FUNCTION_BLOCK FB_MachinePreparation
VAR_INPUT
    // 自动启动协调器或WPF一键整机准备请求。
    // 只受理FALSE→TRUE上升沿。
    bStart : BOOL;

    // Stop、整机故障或流程中止。
    bAbort : BOOL;

    // 故障复位脉冲。
    bReset : BOOL;

    stConfig : ST_MachinePreparationConfig;
END_VAR

VAR_IN_OUT
    aAxes : ARRAY[1..GVL_Constants.cMaxAxisCount]
            OF ST_AxisInterface;
	// 复用MAIN中COM3唯一的自动动作实例。
    // 禁止在准备流程中重新创建FB_GripperAction实例。
    ioGripperAction : FB_GripperAction;
	// 复用MAIN中COM4唯一的自动动作实例。
    ioAdjustGripperAction : FB_GripperAction;

    // COM3夹爪统一接口。
    ioGripper : ST_GripperInterface;
	// COM4调整夹爪统一接口。
    ioAdjustGripper : ST_GripperInterface;
END_VAR

VAR_OUTPUT
    bBusy       : BOOL;
    bDone       : BOOL;
    bError      : BOOL;
    bErrorPulse : BOOL;
    bTimeout    : BOOL;

    uiErrorAxis : UINT;
    udiErrorCode : UDINT;

    eStep : E_MachinePreparationStep :=
        E_MachinePreparationStep.Idle;
END_VAR

VAR
    trigStart : R_TRIG;

    fbReadyTimeout  : TON;
    fbMotionTimeout : TON;
    // 准备私有Tray恢复上下文，每次Start/Stop/Fault均清理。
    eTrayRecoveryStep : E_MachinePreparationStep := E_MachinePreparationStep.TrayWaitForkStable;
    nRecoveryTargetLayer : DINT;
    nRecoveryIndex : DINT;
    nRecoveryMatchCount : DINT;
    bTrayRecoverySelected : BOOL;
    bTrayRecoveryActive : BOOL;
    bRecoveryClassC : BOOL;
    bRecoveryRackPermit : BOOL;
    fbTrayRecoveryTimeout : TON;
    fbTrayReleaseTimeout : TON;
    fbTrayReleaseStable : TON;
    bReleaseConditions : BOOL;
    fbForkStable : TON;
    bForkCandidateInitialized : BOOL;
    bForkCandidate : BOOL;
    bForkStable : BOOL;
    bForkStableValid : BOOL;
    aRecoveryLevelTimer : ARRAY[1..5] OF TON;
    aRecoveryLevelInitialized : ARRAY[1..5] OF BOOL;
    aRecoveryLevelCandidate : ARRAY[1..5] OF BOOL;
    aRecoveryLevelStable : ARRAY[1..5] OF BOOL;
    aRecoveryLevelStableValid : ARRAY[1..5] OF BOOL;
    bRecoveryAllLevelsStable : BOOL;
    bNonTrayStandbyDone : BOOL;

    uiItem : DINT;
    uiAxis : UINT;
    bAllAxesReady : BOOL;

    // 各轴命令已发出锁存
    bTrayXIssued       : BOOL;
    bTrayZIssued       : BOOL;
    bDamperXIssued     : BOOL;
    bDamperYIssued     : BOOL;
    bDamperZIssued     : BOOL;
    bRotationIssued    : BOOL;
    bClampIssued       : BOOL;
    bTurntableIssued   : BOOL;
	bAdjustmentXIssued : BOOL;
	bAdjustmentYIssued : BOOL;
	bAdjustmentZIssued : BOOL;
    bScrewYIssued      : BOOL;
    bScrewZIssued      : BOOL;

    // 各轴到位锁存
    bTrayXDone       : BOOL;
    bTrayZDone       : BOOL;
    bDamperXDone     : BOOL;
    bDamperYDone     : BOOL;
    bDamperZDone     : BOOL;
    bRotationDone    : BOOL;
    bClampDone       : BOOL;
    bTurntableDone   : BOOL;
	bAdjustmentXDone : BOOL;
	bAdjustmentYDone : BOOL;
	bAdjustmentZDone : BOOL;
    bScrewYDone      : BOOL;
    bScrewZDone      : BOOL;
	
	// 机构准备阶段的COM3张开请求。
    // 在MoveToStandby期间保持TRUE，完成后恢复FALSE。
    bGripperOpenExecute : BOOL;

    // COM3夹爪已经张开完成的锁存状态。
    bGripperOpenDone : BOOL;
    bGripperEnableExecute : BOOL;
    bGripperEnableDone : BOOL; // 本次准备Enable写事务完成，不是硬件使能状态
    bGripperEnableReleasePending : BOOL;
    eGripperPreparationCommand : E_GripperCommand;

	// AdjustmentZ处于安全位置后执行COM4闭合。
	bAdjustGripperCloseExecute : BOOL;
	bAdjustGripperCloseDone : BOOL;
    bAdjustGripperEnableExecute : BOOL;
    bAdjustGripperEnableDone : BOOL;
    bAdjustGripperEnableReleasePending : BOOL;
    eAdjustGripperPreparationCommand : E_GripperCommand;
	bAdjustGripperReady : BOOL;
	liAdjustGripperPositionError : LINT;
END_VAR

//==============================================================
// 1. 请求及定时器
//==============================================================
trigStart(CLK := bStart);

fbReadyTimeout(
    IN := (eStep = E_MachinePreparationStep.WaitAxesReady)
          AND NOT bAbort,
    PT := stConfig.tReadyTimeout
);

bErrorPulse := FALSE;
// 默认不请求夹爪动作。
// 只有MoveToStandby步骤尚未完成张开时才置TRUE。
bGripperOpenExecute := FALSE;
bAdjustGripperCloseExecute := FALSE;

bGripperEnableExecute := FALSE;
bAdjustGripperEnableExecute := FALSE;
eGripperPreparationCommand := E_GripperCommand.Open;
eAdjustGripperPreparationCommand := E_GripperCommand.Close;

// COM4准备完成必须由真实状态共同确认，不能只依赖动作完成握手。
liAdjustGripperPositionError :=
    DINT_TO_LINT(ioAdjustGripper.Feedback.diActualPosition)
    - DINT_TO_LINT(ioAdjustGripper.Set.diClosePosition);
IF liAdjustGripperPositionError < 0 THEN
    liAdjustGripperPositionError := -liAdjustGripperPositionError;
END_IF;

bAdjustGripperReady :=
    ioAdjustGripper.State.bSimulationActive
    OR (ioAdjustGripper.Feedback.bOnline
    AND NOT ioAdjustGripper.Feedback.bCommFault
    AND ioAdjustGripper.Feedback.bFaultCodeValid
    AND NOT ioAdjustGripper.Feedback.bFault
    AND NOT ioAdjustGripper.State.bBusy
    AND NOT ioAdjustGripper.Feedback.bBusy
    AND ioAdjustGripper.Feedback.bPositionValid
    AND ioAdjustGripper.Feedback.bCurrentValid
    AND
    (
        liAdjustGripperPositionError
        <= DINT_TO_LINT(ioAdjustGripper.Set.diPositionTolerance)
    )
    AND ioAdjustGripper.Feedback.bClosed);

// 原超时仍保护全部非Tray准备机构；有盘回库由独立总超时保护。
bNonTrayStandbyDone := bDamperXDone AND bDamperYDone AND bDamperZDone
              AND bRotationDone AND bClampDone AND bTurntableDone
              AND bAdjustmentXDone AND bAdjustmentYDone AND bAdjustmentZDone
              AND bScrewYDone AND bScrewZDone
              AND bGripperOpenDone AND bAdjustGripperCloseDone AND bAdjustGripperReady;
fbMotionTimeout(
    IN := (eStep = E_MachinePreparationStep.MoveToStandby)
        AND NOT bAbort
        AND (NOT bNonTrayStandbyDone
            OR (NOT bTrayRecoverySelected AND NOT (bTrayXDone AND bTrayZDone))),
    PT := stConfig.tMotionTimeout
);

//==============================================================
// 2. Preparation命令脉冲默认清除
// 只处理当前十根已明确准备位置的自动流程轴。
//==============================================================
FOR uiItem := LOWER_BOUND(GVL_AxisIndex.AutoProcessAxes, 1) TO UPPER_BOUND(GVL_AxisIndex.AutoProcessAxes, 1) DO
    uiAxis := GVL_AxisIndex.AutoProcessAxes[uiItem];

    aAxes[uiAxis].PreparationCmd.bMoveAbs := FALSE;
    aAxes[uiAxis].PreparationCmd.bMoveRel := FALSE;
    aAxes[uiAxis].PreparationCmd.bJogPos := FALSE;
    aAxes[uiAxis].PreparationCmd.bJogNeg := FALSE;
    aAxes[uiAxis].PreparationCmd.bStop := FALSE;
    aAxes[uiAxis].PreparationCmd.bTorqueControl := FALSE;
END_FOR;


//==============================================================
// 3. 故障复位和Abort
//
// 复位优先于Abort：准备故障会使整机进入Fault，
// 此时bAbort必然为TRUE，因此必须允许复位先清除本FB故障。
//==============================================================
IF bReset THEN
    bBusy := FALSE;
    bDone := FALSE;
    bError := FALSE;
    bTimeout := FALSE;

    uiErrorAxis := 0;
    udiErrorCode := TO_UDINT(E_MachinePreparationErrorCode.None);

    M_ResetProgress();

    eStep := E_MachinePreparationStep.Idle;

ELSIF bAbort THEN
    bBusy := FALSE;
    bDone := FALSE;

    M_ResetProgress();

    // 如果本FB本身已经报错，保持Error状态，
    // 便于故障诊断和后续统一复位。
    IF bError THEN
        eStep := E_MachinePreparationStep.Error;
    ELSE
        eStep := E_MachinePreparationStep.Idle;
    END_IF;

ELSE
    // 仅Done收到新请求时失效旧完成状态；Start撤销不清除本周期Done。
    // 同一扫描复用Idle中的配置检查和M_ResetProgress，不复制准备状态机。
    IF (eStep = E_MachinePreparationStep.Done) AND trigStart.Q THEN
        bDone := FALSE;
        eStep := E_MachinePreparationStep.Idle;
    END_IF;

    CASE eStep OF

        //======================================================
        // 等待启动
        //======================================================
        E_MachinePreparationStep.Idle:
            bBusy := FALSE;

            IF trigStart.Q THEN
                bDone := FALSE;
                bError := FALSE;
                bTimeout := FALSE;
                uiErrorAxis := 0;
                udiErrorCode := TO_UDINT(E_MachinePreparationErrorCode.None);

                M_ResetProgress();

                // 确认十根准备轴均已配置。
                FOR uiItem := 1 TO
                    UPPER_BOUND(GVL_AxisIndex.AutoProcessAxes, 1)
                DO
                    uiAxis :=
                        GVL_AxisIndex.AutoProcessAxes[uiItem];

                    IF NOT GVL_AxisConfig.AxisLimits[
                        uiAxis
                    ].bConfigured THEN
                        bError := TRUE;
                        bErrorPulse := TRUE;
                        uiErrorAxis := uiAxis;
                        udiErrorCode := TO_UDINT(E_MachinePreparationErrorCode.AxisNotConfigured);
                        eStep :=
                            E_MachinePreparationStep.Error;
                        EXIT;
                    END_IF;
                END_FOR;

                IF NOT bError THEN
                    bBusy := TRUE;
                    eStep :=
                        E_MachinePreparationStep.WaitAxesReady;
                END_IF;
            END_IF;


        //======================================================
        // 请求轴使能并等待全部Ready
        //======================================================
        E_MachinePreparationStep.WaitAxesReady:
            bBusy := TRUE;
            bAllAxesReady := TRUE;
            uiErrorAxis := 0;

            FOR uiItem := 1 TO
                UPPER_BOUND(GVL_AxisIndex.AutoProcessAxes, 1)
            DO
                uiAxis :=
                    GVL_AxisIndex.AutoProcessAxes[uiItem];

                IF aAxes[uiAxis].Alarm.bError THEN
                    bError := TRUE;
                    bErrorPulse := TRUE;
                    uiErrorAxis := uiAxis;

                    IF aAxes[uiAxis].Alarm.nErrorID <> 0 THEN
                        udiErrorCode :=
                            aAxes[uiAxis].Alarm.nErrorID;
                    ELSE
                        udiErrorCode := TO_UDINT(E_MachinePreparationErrorCode.AxisAlarmBase)
                            + UINT_TO_UDINT(uiAxis);
                    END_IF;

                    eStep :=
                        E_MachinePreparationStep.Error;
                    EXIT;
                END_IF;

                // Clamping必须先由真实6061确认已经恢复CSP。
                // 若PLC重新激活后驱动仍残留CST，则通过既有MC_Stop
                // 恢复边界请求退出；6061不是8时绝不发布准备运动。
                IF
                    (uiAxis = GVL_AxisIndex.Clamping)
                    AND
                    (
                        aAxes[uiAxis].State.eControlMode
                        <> E_AxisControlMode.Position
                    )
                THEN
                    aAxes[uiAxis].PreparationCmd.bTorqueControl := FALSE;
                    aAxes[uiAxis].PreparationCmd.bStop := TRUE;
                    bAllAxesReady := FALSE;

                    IF uiErrorAxis = 0 THEN
                        uiErrorAxis := uiAxis;
                    END_IF;
                END_IF;

                IF NOT aAxes[uiAxis].State.bReady THEN
                    bAllAxesReady := FALSE;

                    IF uiErrorAxis = 0 THEN
                        uiErrorAxis := uiAxis;
                    END_IF;
                END_IF;
            END_FOR;

            IF eStep <> E_MachinePreparationStep.Error THEN
                IF bAllAxesReady THEN
                    uiErrorAxis := 0;
                    eStep :=
                        E_MachinePreparationStep.MoveToStandby;

                ELSIF fbReadyTimeout.Q THEN
                    bError := TRUE;
                    bTimeout := TRUE;
                    bErrorPulse := TRUE;
                    udiErrorCode := TO_UDINT(E_MachinePreparationErrorCode.AxisReadyTimeout);
                    eStep :=
                        E_MachinePreparationStep.Error;
                END_IF;
            END_IF;


        //======================================================
        // 整机准备位置运动
        //
        // 三条机械分支并行执行：
        // A. TrayX安全后允许TrayZ
        // B. DamperZ安全后允许DamperXY和Rotation
        // C. ScrewdriverZ安全后允许夹紧松开和Y回零，
        //    夹紧松开后允许转台回零
        //======================================================
        E_MachinePreparationStep.MoveToStandby:
            bBusy := TRUE;
			
			//======================================================
			// COM3夹爪准备动作
			//
			// 与DamperZ抬升同时启动，不需要等待DamperZ到位。
			// bExecute保持TRUE，直到FB_GripperAction返回Done。
			//======================================================
            // 同一路复用唯一Action：Enable完成后FALSE释放，Idle后才发位置动作。
            IF NOT bGripperEnableDone THEN
                eGripperPreparationCommand := E_GripperCommand.Enable;
                bGripperEnableExecute := TRUE;
                IF ioGripperAction.bError THEN
                    bGripperEnableExecute := FALSE;
                    bError := TRUE;
                    bErrorPulse := TRUE;
                    uiErrorAxis := 0;
                    udiErrorCode := TO_UDINT(E_MachinePreparationErrorCode.DamperGripperEnableFailed);
                    // 具体底层原因仍保留在Action/AutoFeedback中。
                    eStep := E_MachinePreparationStep.Error;
                ELSIF ioGripperAction.bDone THEN
                    bGripperEnableDone := TRUE;
                    bGripperEnableReleasePending := TRUE;
                    bGripperEnableExecute := FALSE;
                END_IF;
            ELSIF bGripperEnableReleasePending THEN
                IF ioGripperAction.eStep = E_GripperActionStep.Idle THEN
                    bGripperEnableReleasePending := FALSE;
                END_IF;
            ELSIF NOT bGripperOpenDone THEN
                bGripperOpenExecute := TRUE;
			
				// FB_GripperAction在MAIN中的调用结果会跨扫描周期更新。
				IF ioGripperAction.bError THEN
					// COM3张开失败，机构准备失败。
					bGripperOpenExecute := FALSE;
			
					bError := TRUE;
					bErrorPulse := TRUE;
					uiErrorAxis := 0; // 夹爪不是NC轴，所以轴号为0。
			
					// 优先保留下层夹爪错误码，便于追踪具体动作失败原因。
					IF ioGripperAction.udErrorCode <> TO_UDINT(E_GripperErrorCode.None) THEN
						udiErrorCode := ioGripperAction.udErrorCode;
					ELSE
						udiErrorCode := TO_UDINT(E_MachinePreparationErrorCode.GripperOpenFailed);
					END_IF;
			
					eStep := E_MachinePreparationStep.Error;
			
				ELSIF ioGripperAction.bDone THEN
					// 张开完成后锁存，避免重复下发Open。
					bGripperOpenDone := TRUE;
					bGripperOpenExecute := FALSE;
				END_IF;
			END_IF;
            // Tray先等待Fork稳定，再执行原无盘路径或A/B/C恢复。
			M_PrepareTray(
				ioAxes := aAxes
			);
            // 其它机构继续保持原有并行准备时序。
            IF NOT bDamperZDone THEN
                bDamperZDone := M_MoveAxisAbsolute(
                    fTarget := stConfig.fDamperZStandby,
                    fVelocity := stConfig.fDamperVelocity,
                    fTolerance := stConfig.fLinearTolerance,
                    uiAxisIndex := GVL_AxisIndex.DamperZ,
                    ioIssued := bDamperZIssued,
                    ioAxis := aAxes[GVL_AxisIndex.DamperZ]
                );
            END_IF;

            IF NOT bScrewZDone THEN
                bScrewZDone := M_MoveAxisAbsolute(
                    fTarget := stConfig.fScrewdriverZSafe,
                    fVelocity := stConfig.fScrewdriverVelocity,
                    fTolerance := stConfig.fLinearTolerance,
                    uiAxisIndex := GVL_AxisIndex.ScrewdriverZ,
                    ioIssued := bScrewZIssued,
                    ioAxis := aAxes[GVL_AxisIndex.ScrewdriverZ]
                );
            END_IF;


            // DamperZ在110mm后，允许XY及旋转轴并行回位。
            IF bDamperZDone THEN
                IF NOT bDamperXDone THEN
                    bDamperXDone := M_MoveAxisAbsolute(
                        fTarget := stConfig.fDamperXStandby,
                        fVelocity := stConfig.fDamperVelocity,
                        fTolerance := stConfig.fLinearTolerance,
                        uiAxisIndex := GVL_AxisIndex.DamperX,
                        ioIssued := bDamperXIssued,
                        ioAxis := aAxes[GVL_AxisIndex.DamperX]
                    );
                END_IF;

                IF NOT bDamperYDone THEN
                    bDamperYDone := M_MoveAxisAbsolute(
                        fTarget := stConfig.fDamperYStandby,
                        fVelocity := stConfig.fDamperVelocity,
                        fTolerance := stConfig.fLinearTolerance,
                        uiAxisIndex := GVL_AxisIndex.DamperY,
                        ioIssued := bDamperYIssued,
                        ioAxis := aAxes[GVL_AxisIndex.DamperY]
                    );
                END_IF;

                IF NOT bRotationDone THEN
                    bRotationDone := M_MoveAxisAbsolute(
                        fTarget :=
                            stConfig.fDamperRotationZero,
                        fVelocity :=
                            stConfig.fDamperRotationVelocity,
                        fTolerance :=
                            stConfig.fRotationTolerance,
                        uiAxisIndex :=
                            GVL_AxisIndex.DamperRotation,
                        ioIssued := bRotationIssued,
                        ioAxis :=
                            aAxes[GVL_AxisIndex.DamperRotation]
                    );
                END_IF;
            END_IF;

			//==============================================================
			// 调整机构准备：
			// COM4先回到配置层定义的闭合位置并确认有效，
			// 随后才允许AdjustmentZ回准备位置；Z到位后，
			// AdjustmentX/Y再同时回到准备位置。
			//==============================================================
            // 同一路复用唯一Action：Enable完成后FALSE释放，Idle后才发位置动作。
            IF NOT bAdjustGripperEnableDone THEN
                eAdjustGripperPreparationCommand := E_GripperCommand.Enable;
                bAdjustGripperEnableExecute := TRUE;
                IF ioAdjustGripperAction.bError THEN
                    bAdjustGripperEnableExecute := FALSE;
                    bError := TRUE;
                    bErrorPulse := TRUE;
                    uiErrorAxis := 0;
                    udiErrorCode := TO_UDINT(E_MachinePreparationErrorCode.AdjustGripperEnableFailed);
                    // 具体底层原因仍保留在Action/AutoFeedback中。
                    eStep := E_MachinePreparationStep.Error;
                ELSIF ioAdjustGripperAction.bDone THEN
                    bAdjustGripperEnableDone := TRUE;
                    bAdjustGripperEnableReleasePending := TRUE;
                    bAdjustGripperEnableExecute := FALSE;
                END_IF;
            ELSIF bAdjustGripperEnableReleasePending THEN
                IF ioAdjustGripperAction.eStep = E_GripperActionStep.Idle THEN
                    bAdjustGripperEnableReleasePending := FALSE;
                END_IF;
            ELSIF NOT bAdjustGripperCloseDone THEN
                bAdjustGripperCloseExecute := TRUE;

				IF ioAdjustGripperAction.bError THEN
					bAdjustGripperCloseExecute := FALSE;
					bError := TRUE;
					bErrorPulse := TRUE;
					uiErrorAxis := 0;

					IF ioAdjustGripperAction.udErrorCode <> TO_UDINT(E_GripperErrorCode.None) THEN
						udiErrorCode := ioAdjustGripperAction.udErrorCode;
					ELSE
						udiErrorCode := TO_UDINT(E_MachinePreparationErrorCode.AdjustGripperCloseFailed);
					END_IF;

					eStep := E_MachinePreparationStep.Error;

				ELSIF ioAdjustGripperAction.bDone AND bAdjustGripperReady THEN
					bAdjustGripperCloseDone := TRUE;
					bAdjustGripperCloseExecute := FALSE;
				END_IF;
			END_IF;

			// COM4闭合到50000并完成全部有效性确认后，AdjustmentZ才允许上升。
			IF bAdjustGripperCloseDone
				AND bAdjustGripperReady
				AND NOT bAdjustmentZDone
			THEN
				bAdjustmentZDone := M_MoveAxisAbsolute(
					fTarget := stConfig.fAdjustmentZStandby,
					fVelocity := stConfig.fAdjustmentVelocity,
					fTolerance := stConfig.fLinearTolerance,
					uiAxisIndex := GVL_AxisIndex.AdjustmentZ,
					ioIssued := bAdjustmentZIssued,
					ioAxis := aAxes[GVL_AxisIndex.AdjustmentZ]
				);
			END_IF;

			IF bAdjustmentZDone THEN
				IF NOT bAdjustmentXDone THEN
					bAdjustmentXDone := M_MoveAxisAbsolute(
						fTarget := stConfig.fAdjustmentXStandby,
						fVelocity := stConfig.fAdjustmentVelocity,
						fTolerance := stConfig.fLinearTolerance,
						uiAxisIndex := GVL_AxisIndex.AdjustmentX,
						ioIssued := bAdjustmentXIssued,
						ioAxis := aAxes[GVL_AxisIndex.AdjustmentX]
					);
				END_IF;
			
				IF NOT bAdjustmentYDone THEN
					bAdjustmentYDone := M_MoveAxisAbsolute(
						fTarget := stConfig.fAdjustmentYStandby,
						fVelocity := stConfig.fAdjustmentVelocity,
						fTolerance := stConfig.fLinearTolerance,
						uiAxisIndex := GVL_AxisIndex.AdjustmentY,
						ioIssued := bAdjustmentYIssued,
						ioAxis := aAxes[GVL_AxisIndex.AdjustmentY]
					);
				END_IF;
			END_IF;

            // ScrewdriverZ到安全高度后：
            // 夹紧轴松开和ScrewdriverY回零并行。
            IF bScrewZDone THEN
                IF NOT bClampDone THEN
                    IF
                        aAxes[GVL_AxisIndex.Clamping].State.eControlMode
                        <> E_AxisControlMode.Position
                    THEN
                        // 6061未确认CSP时只允许执行受控模式恢复。
                        aAxes[GVL_AxisIndex.Clamping].PreparationCmd.bTorqueControl := FALSE;
                        aAxes[GVL_AxisIndex.Clamping].PreparationCmd.bStop := TRUE;
                    ELSE
                        bClampDone := M_MoveAxisAbsolute(
                            fTarget := stConfig.fClampOpenPosition,
                            fVelocity := stConfig.fClampVelocity,
                            fTolerance := stConfig.fLinearTolerance,
                            uiAxisIndex := GVL_AxisIndex.Clamping,
                            ioIssued := bClampIssued,
                            ioAxis := aAxes[GVL_AxisIndex.Clamping]
                        );
                    END_IF;
                END_IF;

                IF NOT bScrewYDone THEN
                    bScrewYDone := M_MoveAxisAbsolute(
                        fTarget := stConfig.fScrewdriverYZero,
                        fVelocity :=
                            stConfig.fScrewdriverVelocity,
                        fTolerance := stConfig.fLinearTolerance,
                        uiAxisIndex :=
                            GVL_AxisIndex.ScrewdriverY,
                        ioIssued := bScrewYIssued,
                        ioAxis :=
                            aAxes[GVL_AxisIndex.ScrewdriverY]
                    );
                END_IF;
            END_IF;


            // 只要求夹紧轴松开到位，即可允许转台回零。
            IF bClampDone AND NOT bTurntableDone THEN
                bTurntableDone := M_MoveAxisAbsolute(
                    fTarget := stConfig.fTurntableZero,
                    fVelocity := stConfig.fTurntableVelocity,
                    fTolerance := stConfig.fRotationTolerance,
                    uiAxisIndex := GVL_AxisIndex.Turntable,
                    ioIssued := bTurntableIssued,
                    ioAxis := aAxes[GVL_AxisIndex.Turntable]
                );
            END_IF;


            // 按本扫描最新完成锁存判断超时，避免回库等待期间
            // 非Tray分支恰好完成却被上一扫描的未完成状态误报。
            bNonTrayStandbyDone := bDamperXDone AND bDamperYDone AND bDamperZDone
                AND bRotationDone AND bClampDone AND bTurntableDone
                AND bAdjustmentXDone AND bAdjustmentYDone AND bAdjustmentZDone
                AND bScrewYDone AND bScrewZDone
                AND bGripperOpenDone AND bAdjustGripperCloseDone AND bAdjustGripperReady;

            // 十根轴全部满足目标位置才发布Done。
            IF (eStep <> E_MachinePreparationStep.Error)
                AND bTrayXDone
                AND bTrayZDone
                AND bDamperXDone
                AND bDamperYDone
                AND bDamperZDone
				AND bGripperOpenDone
                AND bRotationDone
                AND bClampDone
                AND bTurntableDone
				AND bAdjustmentXDone
				AND bAdjustmentYDone
				AND bAdjustmentZDone
				AND bAdjustGripperCloseDone
				AND bAdjustGripperReady
                AND bScrewYDone
                AND bScrewZDone
            THEN
                bBusy := FALSE;
                bDone := TRUE;
                eStep := E_MachinePreparationStep.Done;

            ELSIF (eStep <> E_MachinePreparationStep.Error)
                AND fbMotionTimeout.Q
                AND (NOT bNonTrayStandbyDone OR NOT bTrayRecoverySelected)
            THEN
                bError := TRUE;
                bTimeout := TRUE;
                bErrorPulse := TRUE;
                udiErrorCode := TO_UDINT(E_MachinePreparationErrorCode.StandbyMotionTimeout);

                // 保存第一根尚未到位的轴。
				    // COM3没有完成张开。
				IF NOT bGripperEnableDone THEN
                    uiErrorAxis := 0;
                    udiErrorCode := TO_UDINT(E_MachinePreparationErrorCode.DamperGripperEnableFailed);
                ELSIF NOT bAdjustGripperEnableDone THEN
                    uiErrorAxis := 0;
                    udiErrorCode := TO_UDINT(E_MachinePreparationErrorCode.AdjustGripperEnableFailed);
                ELSIF NOT bGripperOpenDone THEN
					uiErrorAxis := 0;
					udiErrorCode := TO_UDINT(E_MachinePreparationErrorCode.GripperOpenFailed);
				ELSIF NOT bAdjustGripperCloseDone OR NOT bAdjustGripperReady THEN
					uiErrorAxis := 0;
					udiErrorCode := TO_UDINT(E_MachinePreparationErrorCode.AdjustGripperCloseFailed);
                ELSIF NOT bTrayRecoverySelected AND NOT bTrayXDone THEN
                    uiErrorAxis := GVL_AxisIndex.TrayX;
                ELSIF NOT bTrayRecoverySelected AND NOT bTrayZDone THEN
                    uiErrorAxis := GVL_AxisIndex.TrayZ;
                ELSIF NOT bDamperZDone THEN
                    uiErrorAxis := GVL_AxisIndex.DamperZ;
                ELSIF NOT bDamperXDone THEN
                    uiErrorAxis := GVL_AxisIndex.DamperX;
                ELSIF NOT bDamperYDone THEN
                    uiErrorAxis := GVL_AxisIndex.DamperY;
                ELSIF NOT bRotationDone THEN
                    uiErrorAxis := GVL_AxisIndex.DamperRotation;
                ELSIF NOT bScrewZDone THEN
                    uiErrorAxis := GVL_AxisIndex.ScrewdriverZ;
                ELSIF NOT bClampDone THEN
                    uiErrorAxis := GVL_AxisIndex.Clamping;
				ELSIF NOT bAdjustmentZDone THEN
					uiErrorAxis := GVL_AxisIndex.AdjustmentZ;
				ELSIF NOT bAdjustmentXDone THEN
					uiErrorAxis := GVL_AxisIndex.AdjustmentX;
				ELSIF NOT bAdjustmentYDone THEN
					uiErrorAxis := GVL_AxisIndex.AdjustmentY;
                ELSIF NOT bScrewYDone THEN
                    uiErrorAxis := GVL_AxisIndex.ScrewdriverY;
                ELSIF NOT bTurntableDone THEN
                    uiErrorAxis := GVL_AxisIndex.Turntable;
                END_IF;

                eStep := E_MachinePreparationStep.Error;
            END_IF;


        E_MachinePreparationStep.Done:
            bBusy := FALSE;
            bDone := TRUE;


        E_MachinePreparationStep.Error:
            bBusy := FALSE;
            bDone := FALSE;
            bError := TRUE;


        ELSE
            bError := TRUE;
            bErrorPulse := TRUE;
            udiErrorCode := TO_UDINT(E_MachinePreparationErrorCode.InvalidProcessStep);
            eStep := E_MachinePreparationStep.Error;
    END_CASE;
END_IF;
// 当扫描即清理恢复上下文和未提交运动脉冲，诊断保持到既有Reset。
// 实际减速停止/Stop所有权仍由MAIN中既有安全链处理。
IF eStep = E_MachinePreparationStep.Error THEN
    bBusy := FALSE;
    bDone := FALSE;
    M_ResetTrayRecovery();
    FOR uiItem := LOWER_BOUND(GVL_AxisIndex.AutoProcessAxes, 1)
        TO UPPER_BOUND(GVL_AxisIndex.AutoProcessAxes, 1)
    DO
        uiAxis := GVL_AxisIndex.AutoProcessAxes[uiItem];
        aAxes[uiAxis].PreparationCmd.bMoveAbs := FALSE;
        aAxes[uiAxis].PreparationCmd.bMoveRel := FALSE;
        aAxes[uiAxis].PreparationCmd.bJogPos := FALSE;
        aAxes[uiAxis].PreparationCmd.bJogNeg := FALSE;
        aAxes[uiAxis].PreparationCmd.bTorqueControl := FALSE;
    END_FOR;
END_IF;

//==============================================================
// 4. COM3机构准备动作
//
// WaitAxesReady阶段使用FALSE调用一次，使动作FB完成初始化。
// MoveToStandby阶段各自Enable完成并释放Action后执行Open/Close。
// Error或Abort时撤销动作。
// Done阶段不再调用，命令权交还给自动流程协调器。
//==============================================================

// 如果其他准备轴在本周期报错，必须同时撤销夹爪动作。
IF bAbort
    OR (eStep = E_MachinePreparationStep.Error)
THEN
    bGripperOpenExecute := FALSE;
    bAdjustGripperCloseExecute := FALSE;
    bGripperEnableExecute := FALSE;
    bAdjustGripperEnableExecute := FALSE;
END_IF;

IF bAbort
    OR (eStep = E_MachinePreparationStep.WaitAxesReady)
    OR (eStep = E_MachinePreparationStep.MoveToStandby)
    OR (eStep = E_MachinePreparationStep.Error)
THEN
    ioGripperAction(
        bExecute := bGripperEnableExecute OR bGripperOpenExecute,
        eCommand := eGripperPreparationCommand,
        bAllowCloseTargetWithoutGrip := FALSE, // 准备不继承自动取料授权

        // 整机Stop或准备Abort时立即取消夹爪动作。
        bCancel := bAbort,

        tAcceptTimeout := GVL_ProcessConfig.stGripper.tAcceptTimeout,
        tResultTimeout := GVL_ProcessConfig.stGripper.tResultTimeout,

        ioGripper := ioGripper
    );
END_IF;

// COM4与COM3分别复用MAIN中的唯一Action实例；准备阶段拥有COM4命令权。
IF bAbort
    OR (eStep = E_MachinePreparationStep.WaitAxesReady)
    OR (eStep = E_MachinePreparationStep.MoveToStandby)
    OR (eStep = E_MachinePreparationStep.Error)
THEN
    ioAdjustGripperAction(
        bExecute := bAdjustGripperEnableExecute OR bAdjustGripperCloseExecute,
        eCommand := eAdjustGripperPreparationCommand,
        bCancel := bAbort,
        tAcceptTimeout := GVL_ProcessConfig.stGripper.tAcceptTimeout,
        tResultTimeout := GVL_ProcessConfig.stGripper.tResultTimeout,
        ioGripper := ioAdjustGripper
    );
END_IF;

//==============================================================
// 5. 准备状态机拥有命令权时保持十根轴使能
//
// Done后只要请求尚未撤销，继续保持使能，防止自动启动
// 切换到Automatic前出现一个扫描周期的掉使能。
//==============================================================
IF bBusy
    OR
    (
        (eStep = E_MachinePreparationStep.Done)
        AND bStart
    )
THEN
    FOR uiItem := 1 TO
        UPPER_BOUND(GVL_AxisIndex.AutoProcessAxes, 1)
    DO
        uiAxis :=
            GVL_AxisIndex.AutoProcessAxes[uiItem];

        aAxes[uiAxis].PreparationCmd.bEnable := TRUE;
    END_FOR;
END_IF;

METHOD PRIVATE M_MoveAxisAbsolute : BOOL
VAR_INPUT
    fTarget     : LREAL;
    fVelocity   : LREAL;
    fTolerance  : LREAL;
    uiAxisIndex : UINT;
END_VAR

VAR_IN_OUT
    ioIssued : BOOL;
    ioAxis   : ST_AxisInterface;
END_VAR
M_MoveAxisAbsolute := FALSE;

// 本FB已经进入故障后，不再接受后续轴命令。
IF eStep = E_MachinePreparationStep.Error THEN
    RETURN;
END_IF;

// 轴报警。
IF ioAxis.Alarm.bError THEN
    bError := TRUE;
    bErrorPulse := TRUE;
    uiErrorAxis := uiAxisIndex;

    IF ioAxis.Alarm.nErrorID <> 0 THEN
        udiErrorCode := ioAxis.Alarm.nErrorID;
    ELSE
        udiErrorCode :=
            TO_UDINT(E_MachinePreparationErrorCode.AxisAlarmBase) + UINT_TO_UDINT(uiAxisIndex);
    END_IF;

    eStep := E_MachinePreparationStep.Error;
    RETURN;
END_IF;

// 已经进入目标公差并且轴停止，直接认为本轴完成。
// 因此轴原本就在目标位置时不会重复运动。
IF ioAxis.State.bReady
    AND NOT ioAxis.State.bBusy
    AND
    (
        ABS(ioAxis.Data.fActPosition - fTarget)
        <= fTolerance
    )
THEN
    ioIssued := FALSE;
    M_MoveAxisAbsolute := TRUE;
    RETURN;
END_IF;

// 已发出命令后等待位置反馈。
IF ioIssued THEN
    IF ioAxis.State.bCmdRejected
        OR ioAxis.State.bCommandAborted
    THEN
        bError := TRUE;
        bErrorPulse := TRUE;
        uiErrorAxis := uiAxisIndex;
        udiErrorCode :=
            TO_UDINT(E_MachinePreparationErrorCode.AxisCommandFailureBase) + UINT_TO_UDINT(uiAxisIndex);
        eStep := E_MachinePreparationStep.Error;
    END_IF;

    RETURN;
END_IF;

// 只有Ready且当前不在执行其他运动时才发送新命令。
IF NOT ioAxis.State.bReady
    OR ioAxis.State.bBusy
    OR ioAxis.State.bActive
THEN
    RETURN;
END_IF;

ioAxis.PreparationSet.Position.fAbsolutePosition := fTarget;
ioAxis.PreparationSet.Position.fVelocity := fVelocity;

// 0表示使用当前NC默认加减速度。
ioAxis.PreparationSet.Position.fAcceleration := 0.0;
ioAxis.PreparationSet.Position.fDeceleration := 0.0;

// 只保持一个扫描周期。
ioAxis.PreparationCmd.bMoveAbs := TRUE;
ioIssued := TRUE;
END_METHOD

METHOD PRIVATE M_PrepareTray
VAR_IN_OUT
    ioAxes : ARRAY[1..GVL_Constants.cMaxAxisCount] OF ST_AxisInterface;
END_VAR
// 只在MoveToStandby内调用。所有运动继续经M_MoveAxisAbsolute写PreparationCmd。
IF eStep = E_MachinePreparationStep.Error THEN
    RETURN;
END_IF;

// 即使等待传感器，也优先保留Tray底层真实Axis Error ID。
FOR nRecoveryIndex := GVL_AxisIndex.TrayX TO GVL_AxisIndex.TrayZ DO
    IF ioAxes[nRecoveryIndex].Alarm.bError THEN
        bError := TRUE;
        bErrorPulse := TRUE;
        uiErrorAxis := DINT_TO_UINT(nRecoveryIndex);
        IF ioAxes[nRecoveryIndex].Alarm.nErrorID <> 0 THEN
            udiErrorCode := ioAxes[nRecoveryIndex].Alarm.nErrorID;
        ELSE
            udiErrorCode := TO_UDINT(E_MachinePreparationErrorCode.AxisAlarmBase)
                + DINT_TO_UDINT(nRecoveryIndex);
        END_IF;
        eStep := E_MachinePreparationStep.Error;
        RETURN;
    END_IF;
END_FOR;

// Fork双向稳定确认：候选变化先复位，首次稳定前禁止TrayXZ运动。
IF NOT bForkCandidateInitialized
    OR (bForkCandidate <> GVL_IO.bTrayPresentOnFork)
THEN
    bForkCandidate := GVL_IO.bTrayPresentOnFork;
    bForkCandidateInitialized := TRUE;
    bForkStableValid := FALSE;
    fbForkStable(IN := FALSE, PT := stConfig.tTrayDetectStable);
END_IF;
fbForkStable(IN := TRUE, PT := stConfig.tTrayDetectStable);
IF fbForkStable.Q THEN
    bForkStable := bForkCandidate;
    bForkStableValid := TRUE;
END_IF;

// 准备私有DI稳定状态只用于恢复，不访问生产aTray[]或建立Plan。
bRecoveryAllLevelsStable := TRUE;
FOR nRecoveryIndex := LOWER_BOUND(GVL_IO.aTrayLevelDetected, 1)
    TO UPPER_BOUND(GVL_IO.aTrayLevelDetected, 1)
DO
    IF NOT aRecoveryLevelInitialized[nRecoveryIndex]
        OR (aRecoveryLevelCandidate[nRecoveryIndex]
            <> GVL_IO.aTrayLevelDetected[nRecoveryIndex])
    THEN
        aRecoveryLevelCandidate[nRecoveryIndex] := GVL_IO.aTrayLevelDetected[nRecoveryIndex];
        aRecoveryLevelInitialized[nRecoveryIndex] := TRUE;
        aRecoveryLevelStableValid[nRecoveryIndex] := FALSE;
        aRecoveryLevelTimer[nRecoveryIndex](IN := FALSE, PT := stConfig.tTrayDetectStable);
    END_IF;
    aRecoveryLevelTimer[nRecoveryIndex](IN := TRUE, PT := stConfig.tTrayDetectStable);
    IF aRecoveryLevelTimer[nRecoveryIndex].Q THEN
        aRecoveryLevelStable[nRecoveryIndex] := aRecoveryLevelCandidate[nRecoveryIndex];
        aRecoveryLevelStableValid[nRecoveryIndex] := TRUE;
    END_IF;
    bRecoveryAllLevelsStable := bRecoveryAllLevelsStable
        AND aRecoveryLevelStableValid[nRecoveryIndex];
END_FOR;

// 放盘前稳定丢盘优先故障；Release/回准备位时Fork=FALSE属于预期状态。
IF bTrayRecoveryActive
    AND (eTrayRecoveryStep <> E_MachinePreparationStep.TrayReleaseConfirm)
    AND (eTrayRecoveryStep <> E_MachinePreparationStep.TrayReturnX)
    AND (eTrayRecoveryStep <> E_MachinePreparationStep.TrayReturnZ)
    AND bForkStableValid AND NOT bForkStable
THEN
    M_TrayRecoveryFault(eError := E_MachinePreparationErrorCode.TrayRecoveryForkLost);
    RETURN;
END_IF;

// 到Low以后才计时，且两项条件必须同时连续稳定，禁止立即退X。
bReleaseConditions := FALSE;
IF (eTrayRecoveryStep = E_MachinePreparationStep.TrayReleaseConfirm)
    AND (nRecoveryTargetLayer >= LOWER_BOUND(stConfig.aTrayLayer, 1))
    AND (nRecoveryTargetLayer <= UPPER_BOUND(stConfig.aTrayLayer, 1))
THEN
    bReleaseConditions := GVL_IO.aTrayLevelDetected[nRecoveryTargetLayer]
        AND NOT GVL_IO.bTrayPresentOnFork;
END_IF;
fbTrayReleaseStable(IN := bReleaseConditions, PT := stConfig.tTrayDetectStable);
fbTrayReleaseTimeout(
    IN := (eTrayRecoveryStep = E_MachinePreparationStep.TrayReleaseConfirm),
    PT := stConfig.tTrayReleaseConfirmTimeout
);

CASE eTrayRecoveryStep OF
    E_MachinePreparationStep.TrayWaitForkStable:
        IF bForkStableValid THEN
            IF NOT bForkStable THEN
                // 无盘：保留原X先到Lift、Z再到Standby路径。
                eTrayRecoveryStep := E_MachinePreparationStep.TrayNormalX;
            ELSE
                bTrayRecoverySelected := TRUE;
                bTrayRecoveryActive := TRUE;
                bRecoveryClassC := FALSE;
                IF ABS(ioAxes[GVL_AxisIndex.TrayX].Data.fActPosition
                    - stConfig.fTrayRackStationX) <= stConfig.fTrayRecoveryBoundaryTolerance
                THEN
                    // A类：只按Z区间认层，直接到本层Low。
                    eTrayRecoveryStep := E_MachinePreparationStep.TrayRecoveryLow;
                ELSIF ABS(ioAxes[GVL_AxisIndex.TrayX].Data.fActPosition
                    - stConfig.fTrayXStandby) <= stConfig.fTrayRecoveryBoundaryTolerance
                THEN
                    // C类：完全退出料架，只按稳定空层事实选目标。
                    bRecoveryClassC := TRUE;
                    eTrayRecoveryStep := E_MachinePreparationStep.TrayWaitEmptyLayer;
                ELSIF (ioAxes[GVL_AxisIndex.TrayX].Data.fActPosition
                        > MIN(stConfig.fTrayXStandby, stConfig.fTrayRackStationX))
                    AND (ioAxes[GVL_AxisIndex.TrayX].Data.fActPosition
                        < MAX(stConfig.fTrayXStandby, stConfig.fTrayRackStationX))
                THEN
                    // B类：保持当前Z，X先回Rack；同样只按Z区间认层。
                    eTrayRecoveryStep := E_MachinePreparationStep.TrayRecoveryRack;
                ELSE
                    M_TrayRecoveryFault(eError := E_MachinePreparationErrorCode.TrayRecoveryPositionInvalid);
                END_IF;

                IF NOT bRecoveryClassC AND NOT bError THEN
                    nRecoveryMatchCount := 0;
                    FOR nRecoveryIndex := LOWER_BOUND(stConfig.aTrayLayer, 1)
                        TO UPPER_BOUND(stConfig.aTrayLayer, 1)
                    DO
                        IF (ioAxes[GVL_AxisIndex.TrayZ].Data.fActPosition
                                >= stConfig.aTrayLayer[nRecoveryIndex].fLowPosition
                                    - stConfig.fTrayRecoveryBoundaryTolerance)
                            AND (ioAxes[GVL_AxisIndex.TrayZ].Data.fActPosition
                                <= stConfig.aTrayLayer[nRecoveryIndex].fHighPosition
                                    + stConfig.fTrayRecoveryBoundaryTolerance)
                        THEN
                            nRecoveryMatchCount := nRecoveryMatchCount + 1;
                            nRecoveryTargetLayer := nRecoveryIndex;
                        END_IF;
                    END_FOR;
                    IF nRecoveryMatchCount <> 1 THEN
                        M_TrayRecoveryFault(eError := E_MachinePreparationErrorCode.TrayRecoveryPositionInvalid);
                    END_IF;
                END_IF;
            END_IF;
        END_IF;

    E_MachinePreparationStep.TrayWaitEmptyLayer:
        IF bRecoveryAllLevelsStable THEN
            // 只选择一次，从Layer1至Layer5；五层全满禁止运动。
            FOR nRecoveryIndex := LOWER_BOUND(stConfig.aTrayLayer, 1)
                TO UPPER_BOUND(stConfig.aTrayLayer, 1)
            DO
                IF NOT aRecoveryLevelStable[nRecoveryIndex] THEN
                    nRecoveryTargetLayer := nRecoveryIndex;
                    EXIT;
                END_IF;
            END_FOR;
            IF nRecoveryTargetLayer = 0 THEN
                M_TrayRecoveryFault(eError := E_MachinePreparationErrorCode.TrayRecoveryNoEmptyLayer);
            ELSE
                eTrayRecoveryStep := E_MachinePreparationStep.TrayRecoveryHigh;
            END_IF;
        END_IF;

    E_MachinePreparationStep.TrayRecoveryHigh:
        IF M_MoveAxisAbsolute(
            fTarget := stConfig.aTrayLayer[nRecoveryTargetLayer].fHighPosition,
            fVelocity := stConfig.fTrayVelocity,
            fTolerance := stConfig.fLinearTolerance,
            uiAxisIndex := GVL_AxisIndex.TrayZ,
            ioIssued := bTrayZIssued,
            ioAxis := ioAxes[GVL_AxisIndex.TrayZ])
        THEN
            eTrayRecoveryStep := E_MachinePreparationStep.TrayRecoveryRack;
        END_IF;

    E_MachinePreparationStep.TrayRecoveryRack:
        // C类在真正发X运动前再次确认同一目标仍稳定空；不改投。
        bRecoveryRackPermit := TRUE;
        IF bRecoveryClassC AND NOT bTrayXIssued THEN
            bRecoveryRackPermit := aRecoveryLevelStableValid[nRecoveryTargetLayer];
            IF bRecoveryRackPermit AND aRecoveryLevelStable[nRecoveryTargetLayer] THEN
                bRecoveryRackPermit := FALSE;
                M_TrayRecoveryFault(eError := E_MachinePreparationErrorCode.TrayRecoveryTargetChanged);
            END_IF;
        END_IF;
        IF bRecoveryRackPermit THEN
            IF M_MoveAxisAbsolute(
                fTarget := stConfig.fTrayRackStationX,
                fVelocity := stConfig.fTrayVelocity,
                fTolerance := stConfig.fLinearTolerance,
                uiAxisIndex := GVL_AxisIndex.TrayX,
                ioIssued := bTrayXIssued,
                ioAxis := ioAxes[GVL_AxisIndex.TrayX])
            THEN
                eTrayRecoveryStep := E_MachinePreparationStep.TrayRecoveryLow;
            END_IF;
        END_IF;

    E_MachinePreparationStep.TrayRecoveryLow:
        // A/B不把层传感器当作原仓位占用依据。
        IF M_MoveAxisAbsolute(
            fTarget := stConfig.aTrayLayer[nRecoveryTargetLayer].fLowPosition,
            fVelocity := stConfig.fTrayVelocity,
            fTolerance := stConfig.fLinearTolerance,
            uiAxisIndex := GVL_AxisIndex.TrayZ,
            ioIssued := bTrayZIssued,
            ioAxis := ioAxes[GVL_AxisIndex.TrayZ])
        THEN
            eTrayRecoveryStep := E_MachinePreparationStep.TrayReleaseConfirm;
        END_IF;

    E_MachinePreparationStep.TrayReleaseConfirm:
        IF fbTrayReleaseStable.Q
            AND aRecoveryLevelStableValid[nRecoveryTargetLayer]
            AND aRecoveryLevelStable[nRecoveryTargetLayer]
            AND bForkStableValid AND NOT bForkStable
        THEN
            eTrayRecoveryStep := E_MachinePreparationStep.TrayReturnX;
        ELSIF fbTrayReleaseTimeout.Q THEN
            bTimeout := TRUE;
            M_TrayRecoveryFault(eError := E_MachinePreparationErrorCode.TrayRecoveryReleaseFailed);
        END_IF;

    E_MachinePreparationStep.TrayNormalX,
    E_MachinePreparationStep.TrayReturnX:
        bTrayXDone := M_MoveAxisAbsolute(
            fTarget := stConfig.fTrayXStandby,
            fVelocity := stConfig.fTrayVelocity,
            fTolerance := stConfig.fLinearTolerance,
            uiAxisIndex := GVL_AxisIndex.TrayX,
            ioIssued := bTrayXIssued,
            ioAxis := ioAxes[GVL_AxisIndex.TrayX]);
        IF bTrayXDone THEN
            IF bTrayRecoverySelected THEN
                eTrayRecoveryStep := E_MachinePreparationStep.TrayReturnZ;
            ELSE
                eTrayRecoveryStep := E_MachinePreparationStep.TrayNormalZ;
            END_IF;
        END_IF;

    E_MachinePreparationStep.TrayNormalZ,
    E_MachinePreparationStep.TrayReturnZ:
        bTrayZDone := M_MoveAxisAbsolute(
            fTarget := stConfig.fTrayZStandby,
            fVelocity := stConfig.fTrayVelocity,
            fTolerance := stConfig.fLinearTolerance,
            uiAxisIndex := GVL_AxisIndex.TrayZ,
            ioIssued := bTrayZIssued,
            ioAxis := ioAxes[GVL_AxisIndex.TrayZ]);
        IF bTrayZDone THEN
            bTrayRecoveryActive := FALSE;
            eTrayRecoveryStep := E_MachinePreparationStep.TrayComplete;
        END_IF;

    E_MachinePreparationStep.TrayComplete:
        // Tray Done不替代其它机构Done；最终准备仍由原主状态机汇总。
        bTrayRecoveryActive := FALSE;

    ELSE
        M_TrayRecoveryFault(eError := E_MachinePreparationErrorCode.TrayRecoveryPositionInvalid);
END_CASE;

// 从稳定有盘的分类扫描开始，到X/Lift与Z/Standby完成扫描结束。
fbTrayRecoveryTimeout(
    IN := bTrayRecoveryActive AND NOT bError,
    PT := stConfig.tTrayRecoveryTimeout
);
IF fbTrayRecoveryTimeout.Q AND NOT bError THEN
    bTimeout := TRUE;
    M_TrayRecoveryFault(eError := E_MachinePreparationErrorCode.TrayRecoveryTimeout);
END_IF;
END_METHOD

METHOD PRIVATE M_ResetProgress
VAR_INPUT
END_VAR
M_ResetTrayRecovery();
bTrayXIssued := FALSE;
bTrayZIssued := FALSE;
bDamperXIssued := FALSE;
bDamperYIssued := FALSE;
bDamperZIssued := FALSE;
bRotationIssued := FALSE;
bClampIssued := FALSE;
bTurntableIssued := FALSE;
bScrewYIssued := FALSE;
bScrewZIssued := FALSE;
bAdjustmentXIssued := FALSE;
bAdjustmentYIssued := FALSE;
bAdjustmentZIssued := FALSE;

bTrayXDone := FALSE;
bTrayZDone := FALSE;
bDamperXDone := FALSE;
bDamperYDone := FALSE;
bDamperZDone := FALSE;
bRotationDone := FALSE;
bClampDone := FALSE;
bTurntableDone := FALSE;
bScrewYDone := FALSE;
bScrewZDone := FALSE;
bAdjustmentXDone := FALSE;
bAdjustmentYDone := FALSE;
bAdjustmentZDone := FALSE;

// 清除机构准备阶段的COM3状态。
bGripperOpenExecute := FALSE;
bGripperOpenDone := FALSE;
bGripperEnableExecute := FALSE;
bGripperEnableDone := FALSE;
bGripperEnableReleasePending := FALSE;

// 清除机构准备阶段的COM4状态。
bAdjustGripperCloseExecute := FALSE;
bAdjustGripperCloseDone := FALSE;
bAdjustGripperEnableExecute := FALSE;
bAdjustGripperEnableDone := FALSE;
bAdjustGripperEnableReleasePending := FALSE;
END_METHOD

METHOD PRIVATE M_ResetTrayRecovery
nRecoveryTargetLayer := 0;
nRecoveryMatchCount := 0;
bTrayRecoverySelected := FALSE;
bTrayRecoveryActive := FALSE;
bRecoveryClassC := FALSE;
bRecoveryRackPermit := FALSE;
eTrayRecoveryStep := E_MachinePreparationStep.TrayWaitForkStable;
bTrayXIssued := FALSE;
bTrayZIssued := FALSE;
bTrayXDone := FALSE;
bTrayZDone := FALSE;
bForkCandidateInitialized := FALSE;
bForkCandidate := FALSE;
bForkStable := FALSE;
bForkStableValid := FALSE;
bRecoveryAllLevelsStable := FALSE;
bReleaseConditions := FALSE;
fbForkStable(IN := FALSE, PT := stConfig.tTrayDetectStable);
fbTrayRecoveryTimeout(IN := FALSE, PT := stConfig.tTrayRecoveryTimeout);
fbTrayReleaseTimeout(IN := FALSE, PT := stConfig.tTrayReleaseConfirmTimeout);
fbTrayReleaseStable(IN := FALSE, PT := stConfig.tTrayDetectStable);
FOR nRecoveryIndex := LOWER_BOUND(aRecoveryLevelTimer, 1)
    TO UPPER_BOUND(aRecoveryLevelTimer, 1)
DO
    aRecoveryLevelTimer[nRecoveryIndex](IN := FALSE, PT := stConfig.tTrayDetectStable);
    aRecoveryLevelInitialized[nRecoveryIndex] := FALSE;
    aRecoveryLevelCandidate[nRecoveryIndex] := FALSE;
    aRecoveryLevelStable[nRecoveryIndex] := FALSE;
    aRecoveryLevelStableValid[nRecoveryIndex] := FALSE;
END_FOR;
END_METHOD

METHOD PRIVATE M_TrayRecoveryFault
VAR_INPUT
    eError : E_MachinePreparationErrorCode;
END_VAR
bError := TRUE;
bErrorPulse := TRUE;
uiErrorAxis := 0; // 纯传感器/现场分类错误，不冒充具体轴故障。
udiErrorCode := TO_UDINT(eError);
eStep := E_MachinePreparationStep.Error;
END_METHOD

END_FUNCTION_BLOCK

(* stored: Version 1.1.0.1, ProductVersion 3.1.4026.20
   POU FB_MachinePreparation: Id {fc808fdd-65f0-4d53-b018-734da14a8299}, SpecialFunc None
   Method M_MoveAxisAbsolute: Id {cfaf43b6-532a-449d-9ae3-c6c630b130c4}
   Method M_PrepareTray: Id {b0fb961a-6efa-4506-b0cd-982db79de926}
   Method M_ResetProgress: Id {c29fe135-6b79-4ad5-9d47-96d5f3728157}
   Method M_ResetTrayRecovery: Id {08388bbb-f6b0-495b-935a-39ac6bf3b90e}
   Method M_TrayRecoveryFault: Id {6476248e-3a08-45e4-b899-2f38d308f244} *)
